// TwinCAT 3 PLC project Untitled1
// ProgramVersion: 3.1.4023.0
// libraries:
//   Tc2_Standard, * (Beckhoff Automation GmbH)
//   Tc2_System, * (Beckhoff Automation GmbH)
//   Tc2_Utilities, * (Beckhoff Automation GmbH)
//   Tc3_EventLogger, * (Beckhoff Automation GmbH)
//   Tc3_Module, * (Beckhoff Automation GmbH)
// project tree:
//   / PlcTask.TcTTO
//   POUs/ FB_BaseDevice.TcPOU, FB_Pneumatic.TcPOU, FB_StateManager.TcPOU, F_RemoveProjectName.TcPOU, I_Device.TcIO, I_Pneumatic.TcIO, MAIN.TcPOU, ST_StateHistory.TcDUT, TON_PAUSE.TcPOU
// real-time tasks:
//   TASK PlcTask: cycle T#10ms, priority 20, ADS port 350

CONFIGURATION Untitled1
    RESOURCE PLC ON TwinCAT3
        TASK PlcTask(INTERVAL := T#10ms, PRIORITY := 20);
        PROGRAM MAIN WITH PlcTask : MAIN;
    END_RESOURCE
END_CONFIGURATION

// ---- POUs/ST_StateHistory.TcDUT
TYPE ST_StateHistory :
STRUCT
	state		: INT;
	stateTime	: TIME;
	ts			: TIMESTRUCT;
END_STRUCT
END_TYPE

// ---- POUs/I_Device.TcIO
INTERFACE I_Device EXTENDS __SYSTEM.IQueryInterface

PROPERTY busy : BOOl
GET
END_GET
END_PROPERTY

PROPERTY done : BOOl
GET
END_GET
END_PROPERTY

PROPERTY error : BOOl
GET
END_GET
END_PROPERTY

PROPERTY id : DWORD
GET
END_GET
END_PROPERTY

PROPERTY ready : BOOl
GET
END_GET
END_PROPERTY

METHOD reset : BOOL
VAR_INPUT
END_VAR
END_METHOD

PROPERTY sid : STRING(255)
GET
END_GET
END_PROPERTY

END_INTERFACE

// ---- POUs/I_Pneumatic.TcIO
INTERFACE I_Pneumatic EXTENDS I_Device

METHOD cancel : BOOL
VAR_INPUT
END_VAR
END_METHOD

METHOD doWait : BOOL
VAR_INPUT
END_VAR
END_METHOD

METHOD doWork : BOOL
VAR_INPUT
END_VAR
END_METHOD

PROPERTY isWait : BOOL
GET
END_GET
END_PROPERTY

PROPERTY isWork : BOOL
GET
END_GET
END_PROPERTY

PROPERTY waitText : STRING(255)
GET
END_GET
SET
END_SET
END_PROPERTY

PROPERTY workText : STRING(255)
GET
END_GET
SET
END_SET
END_PROPERTY

END_INTERFACE

// ---- POUs/MAIN.TcPOU
PROGRAM MAIN
VAR
	pneuma: FB_Pneumatic(enDB := FALSE);
	state: INT;
END_VAR


pneuma();

CASE state OF
	5:
		IF pneuma.doWait() THEN
			state := 0;
		END_IF
	10:
		IF pneuma.doWork() THEN
			state := 0;
		END_IF
END_CASE

END_PROGRAM

// ---- POUs/FB_Pneumatic.TcPOU
FUNCTION_BLOCK FB_Pneumatic EXTENDS FB_BaseDevice IMPLEMENTS I_Pneumatic
VAR_INPUT
	waitDelay			: TIME := T#50MS;
	workDelay			: TIME := T#50MS;
	waitItl				: BOOL := TRUE;
	workItl				: BOOL := TRUE;
END_VAR
VAR_OUTPUT
END_VAR
VAR
	_enDB				: BOOL;
	_workText			: STRING(255) := 'Work';
	_waitText			: STRING(255) := 'Wait';
	_workUnMapped		: BOOL;
	_waitUnMapped		: BOOL;
	_first				: BOOL := TRUE;

	workProx	AT %I*	: BOOL;
	waitProx	AT %I*	: BOOL;
	goWork		AT %Q*	: BOOL;
	goWait		AT %Q*	: BOOL;
	goWorkTm			: TON_PAUSE;
	goWaitTm			: TON_PAUSE;
	inWorkTm			: TON;
	inWaitTm			: TON;
	isWorkTrig			: R_TRIG;
	isWaitTrig			: R_TRIG;
	isTempCancel		: BOOL;
	wasWork				: BOOL;
	wasWait				: BOOL;
	tt					: INT;
	avg					: ARRAY [1..2] OF LREAL;
	lastQry				: TIME;
END_VAR
VAR CONSTANT
	cmdWait				: STRING(255) := 'insert into pneumatics (ts, device, direction, time) values (now(), $'%s$', $'wait$', %d);';
	cmdWork				: STRING(255) := 'insert into pneumatics (ts, device, direction, time) values (now(), $'%s$', $'work$', %d);';
	qryGet				: STRING(255) := 'select avg(time) from pneumatics where device = $'%s$' and ts > now() - interval $'30 days$' group by direction order by direction;';
END_VAR

///////////////////////////////////////////////////////////////////////////////
// FB_Pneumatic
//
// v1.0.0
//
///////////////////////////////////////////////////////////////////////////////

inWorkTm(IN := work, PT := workDelay);
inWaitTm(IN := wait, PT := waitDelay);

CASE state OF
	0:
		first();

		{IF defined (variable: DB.Ack)}
		IF _enDB AND_THEN TIME() - lastQry > T#24H AND_THEN NOT DB.Ack.busy THEN
			// Start it here to trigger its busy so no one else can take it
			DB.Ack.execRet1(ADR(qryGet), ADR(avg), SIZEOF(avg), F_STRING(_sid));
			state := 10;
		ELSE
			state := 1000;
		END_IF
		{ELSE}
		state := 1000;
		{END_IF}
	10:
		{IF defined (variable: DB.Ack)}
		// Continue running until result
		IF DB.Ack.done OR_ELSE DB.Ack.error THEN
			// If fails the avg will stay at 0 and will not be used
			lastQry := TIME();
			state := 1000;
		END_IF
		{ELSE}
		state := 1000;
		{END_IF}
	1000:
		isWorkTrig(CLK := isWork);
		IF isWorkTrig.Q AND goWork THEN
			tt := TO_INT(goWorkTm.ET);
			{IF defined (variable: DB.Pool)}
			IF _enDb THEN
				DB.Pool.exec2(ADR(cmdWork), TRUE, F_STRING(_sid), F_INT(tt));
				IF TO_LREAL(goWorkTm.ET) > avg[2] * 1.3 AND avg[2] > 0 THEN
					msg.CreateEx(TC_EVENTS.PneumaticEventClass.WorkSlow, 0);
					msg.ipArguments.Clear().AddInt(TO_INT(goWorkTm.ET)).AddLReal(TO_INT(avg[2]));
					msg.Send(0);
				END_IF
			END_IF
			{END_IF}
		END_IF
		isWaitTrig(CLK := isWait);
		IF isWaitTrig.Q AND goWait THEN
			tt := TO_INT(goWaitTm.ET);
			{IF defined (variable: DB.Pool)}
			IF _enDb THEN
				DB.Pool.exec2(ADR(cmdWait), TRUE, F_STRING(_sid), F_INT(tt));
				IF TO_LREAL(goWaitTm.ET) > avg[1] * 1.3 AND avg[1] > 0 THEN
					msg.CreateEx(TC_EVENTS.PneumaticEventClass.WaitSlow, 0);
					msg.ipArguments.Clear().AddInt(TO_INT(goWaitTm.ET)).AddLReal(TO_INT(avg[1]));
					msg.Send(0);
				END_IF
			END_IF
			{END_IF}
		END_IF
		IF wait AND work THEN
			alarm(TC_EVENTS.PneumaticEventClass.DoubleSensor);
		END_IF
		goWorkTm(IN := goWork, PAUSE := isWork, PT := T#5S);
		goWaitTm(IN := goWait, PAUSE := isWait, PT := T#5S);
		IF goWorkTm.Q THEN
			IF goWorkTm.CNT > 1 THEN
				alarm(TC_EVENTS.PneumaticEventClass.WorkFlickerTimeout);
			ELSE
				alarm(TC_EVENTS.PneumaticEventClass.WorkTimeout);
			END_IF
		END_IF
		IF goWaitTm.Q THEN
			IF goWaitTm.CNT > 1 THEN
				alarm(TC_EVENTS.PneumaticEventClass.WaitFlickerTimeout);
			ELSE
				alarm(TC_EVENTS.PneumaticEventClass.WaitTimeout);
			END_IF
		END_IF
	-1:
		cancel();
	-1000:
		cancel();
		state := 0;
END_CASE

SUPER^();

{attribute 'monitoring' := 'variable'}
PROPERTY busy : BOOL
GET

busy := (goWork AND NOT isWork) OR (goWait AND NOT isWait);
END_GET
END_PROPERTY

METHOD cancel : BOOL
VAR_INPUT
END_VAR

goWait := goWork := FALSE;
cancel := TRUE;
END_METHOD

{attribute 'monitoring' := 'variable'}
PROPERTY done : BOOL
GET

done := (goWork AND isWork) OR (goWait AND isWait);
END_GET
END_PROPERTY

METHOD doWait : BOOL
VAR_INPUT
END_VAR

IF ready AND waitItl THEN
	goWait := TRUE;
	goWork := FALSE;
END_IF
doWait := isWait;
END_METHOD

METHOD doWork : BOOL
VAR_INPUT
END_VAR

IF ready AND workItl THEN
	goWork := TRUE;
	goWait := FALSE;
END_IF
doWork := isWork;
END_METHOD

METHOD FB_init : BOOL
VAR_INPUT
	bInitRetains	: BOOL; // if TRUE, the retain variables are initialized (warm start / cold start)
	bInCopyCode		: BOOL;  // if TRUE, the instance afterwards gets moved into the copy code (online change)
	enDB			: BOOL;
END_VAR

_enDB := enDB;
lastQry := TIME() - T#23H59M;
END_METHOD

METHOD PROTECTED first : BOOL
VAR_INPUT
END_VAR

// Cannot be put into the FB_init method since it happens before
// cyclic cycle and mapping status is not synch yet
IF _first THEN
	_workUnMapped := F_GetMappingStatus(ADR(workProx), SIZEOF(workProx)) = 0;
	_waitUnMapped := F_GetMappingStatus(ADR(waitProx), SIZEOF(waitProx)) = 0;
	_first := FALSE;
END_IF
END_METHOD

{attribute 'monitoring' := 'variable'}
PROPERTY isWait : BOOL
GET

isWait := inWaitTm.Q;
END_GET
END_PROPERTY

{attribute 'monitoring' := 'variable'}
PROPERTY isWork : BOOL
GET

isWork := inWorkTm.Q;
END_GET
END_PROPERTY

METHOD tempCancel : BOOL
VAR_INPUT
END_VAR

IF NOT isTempCancel THEN
	wasWork := goWork;
	wasWait := goWait;
	isTempCancel := TRUE;
END_IF
cancel();
END_METHOD

METHOD tempContinue : BOOL
VAR_INPUT
END_VAR

IF isTempCancel THEN
	goWork := wasWork;
	goWait := wasWait;
	isTempCancel := FALSE;
END_IF
END_METHOD

{attribute 'monitoring' := 'variable'}
PROPERTY PROTECTED wait : BOOL
GET

wait := waitProx OR_ELSE (_waitUnMapped AND goWait);
END_GET
END_PROPERTY

PROPERTY waitText : STRING(255)
GET

waitText := _waitText;
END_GET
SET

_waitText := waitText;
END_SET
END_PROPERTY

{attribute 'monitoring' := 'variable'}
PROPERTY PROTECTED work : BOOL
GET

work := workProx OR_ELSE (_workUnMapped AND goWork);
END_GET
END_PROPERTY

PROPERTY workText : STRING(255)
GET

workText := _workText;
END_GET
SET

_workText := workText;
END_SET
END_PROPERTY

END_FUNCTION_BLOCK

// ---- POUs/FB_BaseDevice.TcPOU
{attribute 'reflection'}
FUNCTION_BLOCK FB_BaseDevice IMPLEMENTS I_Device
VAR_INPUT
	safetyOK			: BOOL := TRUE;
END_VAR
VAR_OUTPUT
END_VAR
VAR
	{attribute 'instance-path'} 
    {attribute 'noinit'} 
    _sid				: STRING(255);
	_id					: WORD;
	_it					: I_Device;

	state				: INT;
	SM					: FB_StateManager;
	staleResetTm		: TON;
	staleResetTime		: TIME := T#1S;
	textState			: STRING(255) := 'Waiting for ready';

	msg					: FB_TcMessage;
END_VAR

///////////////////////////////////////////////////////////////////////////////
// FB_BaseDevice
//
// v1.0.0
//
// busy: Defaults to false
// done: Defaults to false
// error: Defaults to state < 0
// ready: Defaults to state >= 1000
///////////////////////////////////////////////////////////////////////////////

SM(state := state);
staleResetTm(IN := state <= -1000, PT := staleResetTime);

CASE state OF
	0:
		textState := 'Waiting for ready';
	999:
		textState := 'Idle';
	1000:
		textState := 'Running';
	-1:
		textState := 'Error';
	-1000:
		textState := 'Resetting';
END_CASE

METHOD PROTECTED FINAL alarm : BOOL
VAR_INPUT
	evt	: TcEventEntry;
END_VAR

alarm := alarmJson(evt, '');
END_METHOD

METHOD PROTECTED FINAL alarmAds : BOOL
VAR_INPUT
	errorId	: UDINT;
END_VAR

state := -1;
msg.Create(TC_EVENT_CLASSES.AdsEventClass, errorId, TcEventSeverity.Error, 0);
msg.Send(0);
END_METHOD

METHOD PROTECTED FINAL alarmJson : BOOL
VAR_INPUT
	evt	: TcEventEntry;
	str	: STRING(255);
END_VAR

state := -1;

msg.CreateEx(evt, 0);
IF len(str) > 0 THEN
	msg.SetJsonAttribute(str);
END_IF

msg.Send(0);
END_METHOD

{attribute 'monitoring' := 'variable'}
PROPERTY busy : BOOL
GET

busy := FALSE;
END_GET
END_PROPERTY

{attribute 'monitoring' := 'variable'}
PROPERTY done : BOOL
GET

done := FALSE;
END_GET
END_PROPERTY

{attribute 'monitoring' := 'variable'}
PROPERTY error : BOOL
GET

error := state < 0;
END_GET
END_PROPERTY

METHOD FB_init : BOOL
VAR_INPUT
	bInitRetains : BOOL; // if TRUE, the retain variables are initialized (warm start / cold start)
	bInCopyCode : BOOL;  // if TRUE, the instance afterwards gets moved into the copy code (online change)
END_VAR

_sid := F_RemoveProjectName(_sid);
_id := F_DATA_TO_CRC16_CCITT(ADR(_sid), TO_UDINT(len(_sid)), 0);
_it := THIS^;
{IF defined (variable: DH)}
DH.pushDevice(_sid, THIS);
{END_IF}

// Call release to help if the FB is made persistent
msg.Release();
END_METHOD

{attribute 'monitoring' := 'variable'}
PROPERTY id : DWORD
GET

id := _id;
END_GET
END_PROPERTY

METHOD PROTECTED FINAL message : BOOL
VAR_INPUT
	evt	: TcEventEntry;
END_VAR

message := messageJson(evt, '');
END_METHOD

METHOD PROTECTED FINAL messageJson : BOOL
VAR_INPUT
	evt	: TcEventEntry;
	str	: STRING(255);
END_VAR

msg.CreateEx(evt, 0);
IF len(str) > 0 THEN
	msg.SetJsonAttribute(str);
END_IF
msg.Send(0);
END_METHOD

{attribute 'monitoring' := 'variable'}
PROPERTY ready : BOOL
GET

ready := state >= 1000;
END_GET
END_PROPERTY

METHOD FINAL reset : BOOL
VAR_INPUT
END_VAR

IF state > -1000 OR staleResetTm.Q THEN
	staleResetTm(IN := FALSE);
	state := -1000;
END_IF
reset := ready;
END_METHOD

{attribute 'monitoring' := 'variable'}
PROPERTY FINAL sid : STRING(255)
GET

sid := _sid;
END_GET
END_PROPERTY

END_FUNCTION_BLOCK

// ---- POUs/FB_StateManager.TcPOU
FUNCTION_BLOCK FB_StateManager
VAR_IN_OUT
	state		: INT;
END_VAR
VAR
	data		: ARRAY [1..25] OF ST_StateHistory;
	prevState	: INT;
	stateStart	: TIME;
END_VAR

///////////////////////////////////////////////////////////////////////////////
// FB_StateManager
//
// v1.0.0
//
// The first few state changes will have UTC time until the tz info is fetched.
// Users Logger to get timezone information
///////////////////////////////////////////////////////////////////////////////

IF state <> prevState THEN
	data[1].stateTime := stateTime;
	MEMCPY(ADR(data) + SIZEOF(ST_StateHistory), ADR(data), SIZEOF(data) - SIZEOF(ST_StateHistory));
	data[1].state := state;
	data[1].stateTime := T#0MS;
	prevState := state;

	// If available set, otherwise too expensive to compute
	{IF defined (variable: SysTime)}
	data[1].ts := SysTime.systemTime;
	{END_IF}

	// If available use, but compute if not as needed for output
	// Setting globally can allow fairly significant savings
	{IF defined (variable: CurTime)}
	stateStart := CurTime;
	{ELSE}
	stateStart := TIME();
	{END_IF}
END_IF

METHOD FB_init : BOOL
VAR_INPUT
	bInitRetains : BOOL; // if TRUE, the retain variables are initialized (warm start / cold start)
	bInCopyCode : BOOL;  // if TRUE, the instance afterwards gets moved into the copy code (online change)
END_VAR

stateStart := TIME();
END_METHOD

PROPERTY stateTime : TIME
GET

{IF defined (variable: CurTime)}
stateTime := CurTime - stateStart;
{ELSE}
stateTime := TIME() - stateStart;
{END_IF}
END_GET
END_PROPERTY

END_FUNCTION_BLOCK

// ---- POUs/F_RemoveProjectName.TcPOU
FUNCTION F_RemoveProjectName : STRING(255)
VAR_INPUT
	path	: STRING(255);
END_VAR

///////////////////////////////////////////////////////////////////////////////
// F_RemoveProjectName
//
// v1.0.0
///////////////////////////////////////////////////////////////////////////////

F_RemoveProjectName := DELETE(path, LEN(TwinCAT_SystemInfoVarList._AppInfo.ProjectName) + FIND(path, TwinCAT_SystemInfoVarList._AppInfo.ProjectName), 1);
F_RemoveProjectName := F_ToLCase(F_RemoveProjectName);

END_FUNCTION

// ---- POUs/TON_PAUSE.TcPOU
FUNCTION_BLOCK TON_PAUSE
VAR_INPUT
	IN : BOOL;
	PT : TIME;
	PAUSE : BOOL;
END_VAR
VAR_OUTPUT
	Q : BOOL;
	ET : TIME;
	CNT : UINT;
END_VAR
VAR
	trig : R_TRIG;
	tm : TON;
	pauseTime : TIME;
END_VAR

///////////////////////////////////////////////////////////////////////////////
// TON_PAUSE
//
// v1.0.0
//
///////////////////////////////////////////////////////////////////////////////

IF NOT IN THEN
    pauseTime := T#0S;
	CNT := 0;
END_IF

trig(CLK := IN AND PAUSE);
IF trig.Q THEN
    pauseTime := pauseTime + tm.ET;
	CNT := CNT + 1;
END_IF

IF IN AND pauseTime >= PT THEN
	Q := TRUE;
	ET := PT;
ELSE
	tm(IN := IN AND NOT PAUSE, PT := PT - pauseTime);
	Q := tm.Q;
	ET := pauseTime + tm.ET;
END_IF

END_FUNCTION_BLOCK
